FUNCTION_BLOCK AnalogInput_Status (* Composite Function Block Type *)
  (* Standard: 61499-2 *)
  (* Version 0.0, 8/31/2022, SESA583220, Schneider Electric, template *)
  PACKAGE SE.Nereda;
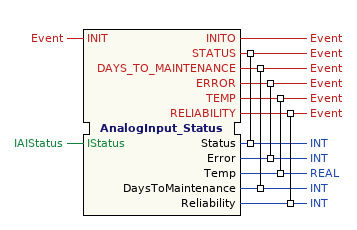
  EVENT_INPUT
    INIT; (* Initializes the symbolic link data destination FB with N (1 <= N <= 16) variables *)
  END_EVENT
  EVENT_OUTPUT
    INITO; (* Initialization Confirm *)
    STATUS WITH Status; (* Confirmation of an explicit or implicit data read request *)
    DAYS_TO_MAINTENANCE WITH DaysToMaintenance; (* Confirmation of an explicit or implicit data read request *)
    ERROR WITH Error; (* Confirmation of an explicit or implicit data read request *)
    TEMP WITH Temp; (* Confirmation of an explicit or implicit data read request *)
    RELIABILITY WITH Reliability; (* Confirmation of an explicit or implicit data read request *)
  END_EVENT
  VAR_OUTPUT
    Status : INT; (* Current value(i) in the named variable array element *)
    Error : INT; (* Current value(i) in the named variable array element *)
    Temp : REAL; (* Current value(i) in the named variable array element *)
    DaysToMaintenance : INT; (* Current value(i) in the named variable array element *)
    Reliability : INT; (* Current value(i) in the named variable array element *)
  END_VAR
  SOCKETS
    IStatus : IAIStatus;
  END_SOCKETS
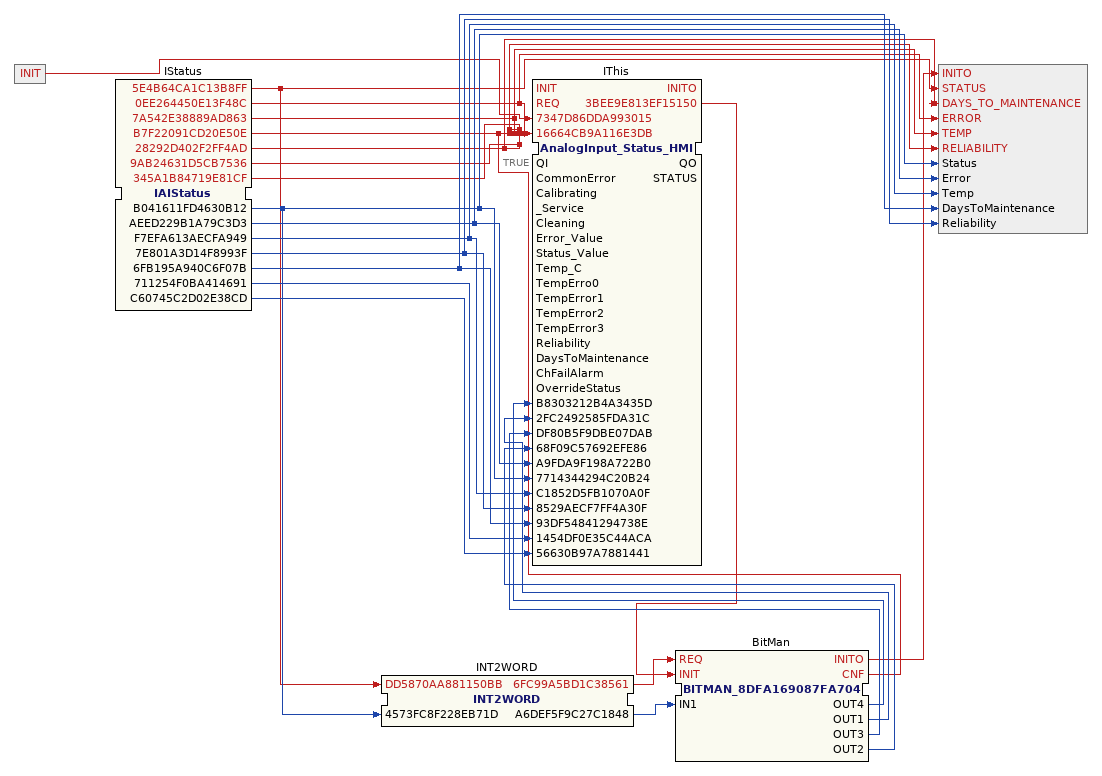
  (* 01 - FUNCTIONNAL INPUT INTERFACE *)
  (* 06 - HMI INTERFACE *)
  (* 02 - FUNCTIONNAL OUTPUT INTERFACE *)
  (* 05 - LOGIC *)
  FBS
    IThis : AnalogInput_Status_HMI(QI := TRUE);
    BitMan : BITMAN_8DFA169087FA704; {SET_ATTRIBUTE(Configuration.GenericFBType.InterfaceParams, Runtime.Standard#CNTIN:=1;CNTOUT:=4;IN${CNTIN$}:WORD;OUT${CNTOUT$}:BOOL,BOOL,BOOL,BOOL)}
    INT2WORD : INT2WORD;
  END_FBS
  EVENT_CONNECTIONS
    BitMan.INITO TO INITO;
    IStatus.5E4B64CA1C13B8FF TO STATUS;
    IStatus.5E4B64CA1C13B8FF TO INT2WORD.DD5870AA881150BB;
    IStatus.0EE264450E13F48C TO ERROR;
    IStatus.7A542E38889AD863 TO TEMP;
    IStatus.B7F22091CD20E50E TO RELIABILITY;
    IStatus.28292D402F2FF4AD TO DAYS_TO_MAINTENANCE;
    INT2WORD.6FC99A5BD1C38561 TO BitMan.REQ;
    INIT TO IThis.7347D86DDA993015;
    BitMan.CNF TO IThis.16664CB9A116E3DB;
    IStatus.0EE264450E13F48C TO IThis.16664CB9A116E3DB;
    IStatus.7A542E38889AD863 TO IThis.16664CB9A116E3DB;
    IStatus.B7F22091CD20E50E TO IThis.16664CB9A116E3DB;
    IStatus.28292D402F2FF4AD TO IThis.16664CB9A116E3DB;
    IStatus.9AB24631D5CB7536 TO IThis.16664CB9A116E3DB;
    IStatus.345A1B84719E81CF TO IThis.16664CB9A116E3DB;
    IThis.3BEE9E813EF15150 TO BitMan.INIT;
  END_CONNECTIONS
  DATA_CONNECTIONS
    IStatus.B041611FD4630B12 TO Status;
    IStatus.B041611FD4630B12 TO INT2WORD.4573FC8F228EB71D;
    IStatus.AEED229B1A79C3D3 TO Error;
    IStatus.F7EFA613AECFA949 TO Temp;
    IStatus.7E801A3D14F8993F TO Reliability;
    IStatus.6FB195A940C6F07B TO DaysToMaintenance;
    INT2WORD.A6DEF5F9C27C1848 TO BitMan.IN1;
    BitMan.OUT4 TO IThis.B8303212B4A3435D;
    BitMan.OUT1 TO IThis.2FC2492585FDA31C;
    BitMan.OUT3 TO IThis.DF80B5F9DBE07DAB;
    BitMan.OUT2 TO IThis.68F09C57692EFE86;
    IStatus.AEED229B1A79C3D3 TO IThis.A9FDA9F198A722B0;
    IStatus.B041611FD4630B12 TO IThis.7714344294C20B24;
    IStatus.F7EFA613AECFA949 TO IThis.C1852D5FB1070A0F;
    IStatus.7E801A3D14F8993F TO IThis.8529AECF7FF4A30F;
    IStatus.6FB195A940C6F07B TO IThis.93DF54841294738E;
    IStatus.711254F0BA414691 TO IThis.1454DF0E35C44ACA;
    IStatus.C60745C2D02E38CD TO IThis.56630B97A7881441;
  END_CONNECTIONS
END_FUNCTION_BLOCK
